// TIA Portal V19 export
FUNCTION_BLOCK "FlyingCarriage_FB"   // FB112, LAD
TITLE = FLYING SHEAR CARRIAGE
// stored: MemoryReserve 100, SetENOAutomatically false
   VAR_INPUT
      AreaInterface : "AreaInterface";
      ZSI : "udt_ZoneSafetyInterface";
      DSI : "udt_DeviceSafetyInterface";
      Drive { ExternalAccessible := 'False'; ExternalVisible := 'False'; ExternalWritable := 'False'} : "TAx_DriveInterface";
      CIn : "udt_FlyingCarriage_CIn";
      DataIn { ExternalAccessible := 'False'; ExternalVisible := 'False'; ExternalWritable := 'False'} : Struct
         Pb_Bkw : Bool;
         Pb_Fwd : Bool;
         Pb_Pos : Bool;
         Pb_Zero : Bool;
         Pb_PresetPos : Bool;
         Fbk_Fan : Bool;
      END_STRUCT;
      Config { ExternalAccessible := 'False'; ExternalVisible := 'False'; ExternalWritable := 'False'} : "udt_FlyingCarriage_Config";
   END_VAR
   VAR_OUTPUT
      MachineInterface : "MachineInterface";
      DataOut : Struct
         Fan : Bool;
         LP_ZeroOK : Bool;
      END_STRUCT;
   END_VAR
   VAR_IN_OUT
      TO_Carriage : TO_SynchronousAxis;
      TO_Master : TO_PositioningAxis;
      TO_ZeroChk : TO_MeasuringInput;
      Parameter : "udt_FlyingCarriage_Parameter";
      FsParameter : "udt_FsParameter";
   END_VAR
   VAR
      Warning : Struct
         NotAutReady : Bool := FALSE;
         ZeroChkRequest : Bool := FALSE;
         Axis : "TAx_Warnings";
      END_STRUCT;
      Alarm : Struct
         NotHomed : Bool := FALSE;
         ZeroChkFailed : Bool := FALSE;
         ZeroChk_NotCatched : Bool := FALSE;
         ZeroChk_NotReleased : Bool := FALSE;
         TargetPosition_OutOfRange : Bool := FALSE;
         Axis : "TAx_Alarms";
         ZeroChk : "TMeasuring_Alarms";
         Fan : "MotorAlr";
      END_STRUCT;
      Diag : Struct
         Ax : "TO_Diagnostic";
         ZeroChk : "TO_Diagnostic";   // 0 = No Msg; 1=Warning; 2= Fault
      END_STRUCT;
      COut : Struct
         Infeed_ReqON : Bool := FALSE;
         CtrlSafe : Bool := FALSE;
         Ax_InOperation : Bool := FALSE;
         Standstill : Bool := FALSE;
         CheckNext_Minus : Bool := FALSE;
         CheckNext_Plus : Bool := FALSE;
         PositioningDone : Bool := FALSE;
         InSynch : Bool := FALSE;
         ActualTargetPosAx : LReal := 0.0;
      END_STRUCT;
      HMI : Struct
         Pb_PresetPos : Bool := FALSE;
         PresetPosValue : LReal := 0.0;
         LastPositionDetect : LReal := 0.0;
         ManPosTarget : LReal;
         PositionNorm : Real;   // Normalized between 0.0 - 1.0
      END_STRUCT;
      Ax { S7_SetPoint := 'True'} : "FlyingShearAxis";
      MeasInp_ZeroChk { S7_SetPoint := 'True'} : "MeasuringInput";
      M_MotorFan : "Motor";
      tonDelayFanOff { S7_SetPoint := 'True'} : IEC_TIMER;
      tonDelayNoPendingCommands : IEC_TIMER;
      Sts : Struct
         IsStandstill : Bool;
         AlarmsPresence : Bool;
         WarningsPresence : Bool;
         DriveMessagesPresence : Bool;
         AxisMessagePresence : Bool;
         InOperatin : Bool;
         DriveParReadWriteDone : Bool;
         DriveMessagesReadDone : Bool;
         Gen_Condition : Bool;
         Bkw_Condition : Bool;
         Fwd_Condition : Bool;
         NoManCmd : Bool;
         Positioning_Condition : Bool;
         MotionRequestInNegativeDirection : Bool;
         MotionRequestInPositiveDirection : Bool;
         InPosition : Bool;
         AtHomePosition : Bool;
         Target_PosAx : LReal;
         MissingToTarget : LReal;
         ActualLimitMinus : LReal;
         ActualLimitPlus : LReal;
         ZeroChk_LastPositionDetect : LReal;
         ZeroChk_MeasInLastID : UInt;
      END_STRUCT;
      Ctrl : Struct
         RstAlarms : Bool;
         SafeMotion : Bool;
         StopDueDoorOpeningRequest : Bool;
         StopSafe : Bool;
         StopInPhase : Bool;
         StopProgrammed : Bool;
         StopAborting : Bool;
         ReadSLSParam : Bool;
         DriveParReadWrite_Exe : Bool;
         DriveMessageRead_Exe : Bool;
         Fan : Bool;
         Man_JogPosBkw : Bool;
         Man_JogPosFwd : Bool;
         Man_Pos : Bool;
         Man_Zero : Bool;
         Zero_Bkw : Bool;
         Zero_Fwd : Bool;
         Zero_Home : Bool;
         Man_Zero_Bkw : Bool;
         Man_Zero_Fwd : Bool;
         Man_Zero_Home : Bool;
         Man_PresetPosition : Bool;
         Aut_Zero : Bool;
         Aut_PosAbs : Bool;
         Aut_GearPos : Bool;
      END_STRUCT;
      AckRstAlarms : Bool := FALSE;
      Pb_Bkw_PEAux : Bool := FALSE;
      Pb_Fwd_PEAux : Bool := FALSE;
      Pb_Pos_PEAux : Bool := FALSE;
      Pb_Zero_PEAux : Bool := FALSE;
      Pb_PresetPos_PEAux : Bool := FALSE;
      ZeroChk_LastID : UInt := 0;
   END_VAR
   VAR_TEMP
      "NOP" : Bool;
      Pb_Bkw_PositiveEdge : Bool;
      Pb_Fwd_PositiveEdge : Bool;
      Pb_Pos_PositiveEdge : Bool;
      Pb_Zero_PositiveEdge : Bool;
      Pb_PresetPos_PositiveEdge : Bool;
      KP_FromProfilePrg : Real;
      KI_FromProfilePrg : Real;
      Delta_KP : Real;
      Delta_KI : Real;
      Delta_ChkZero : LReal;
      Jerk_Multi : LReal;
      Req : Bool;
   END_VAR
   VAR CONSTANT
      EXTENDED_SAFETY : Bool := FALSE;
      SLS_VEL : LReal := 3.0;
      DEFAULT_KV : LReal := 10.0;
      DEFAULT_KP : Real := 5.0;
      DEFAULT_KI : Real := 10.0;
      PAR_FLT : UInt := 0;
      PAR_ALM : UInt := 1;
      PAR_SLS : UInt := 2;
      PAR_KP : UInt := 3;
      PAR_KI : UInt := 4;
      DPS_IDLE : USInt := 0;
      DPS_REQUEST : USInt := 1;
      DPS_ACTIVE : USInt := 2;
      DPS_DONE : USInt := 10;
      DPS_ERROR : USInt := 11;
   END_VAR
   // MachineInterface.AutReady := FALSE;
   // MachineInterface.Aborting := FALSE;
   // MachineInterface.AckStopInPhase := FALSE;
   // MachineInterface.AckStopProgrammed := FALSE;
   // MachineInterface.MotionsStandStill := TRUE;
   // MachineInterface.AlarmsPresence := FALSE;
   // MachineInterface.WarningPresence := FALSE;
   VAR_TEMP   // added for the SCL form of the ladder/FBD networks
      _w1 : Bool;
      _w2 : Bool;
      _w3 : Bool;
      _w4 : Bool;
      _w5 : Bool;
   END_VAR
BEGIN

REGION Network 1: Push buttons positive edges
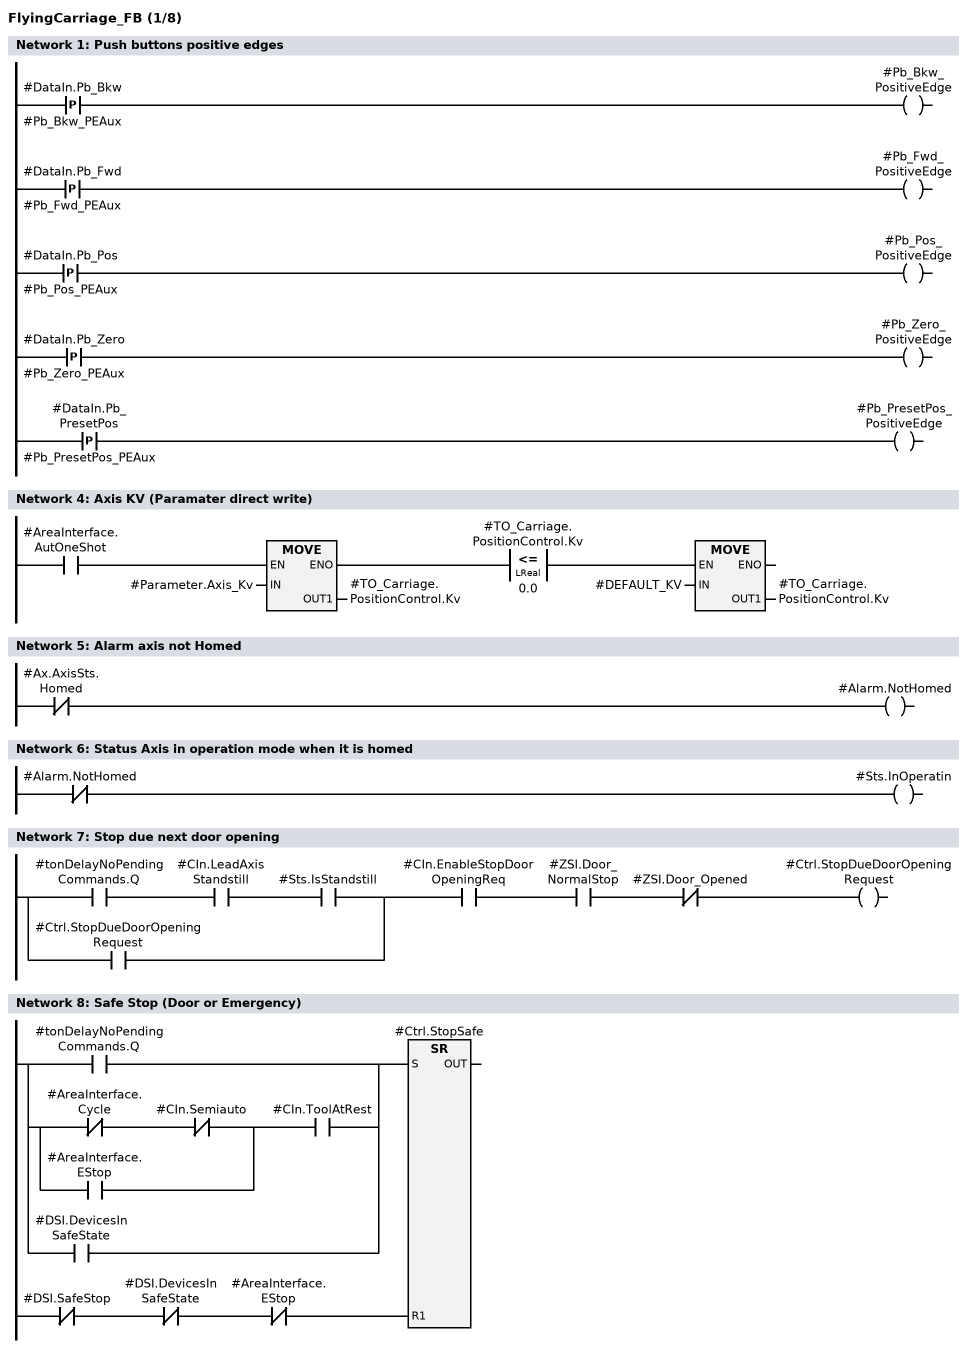
   RUNG wire#powerrail
      P_Contact(operand := #DataIn.Pb_Bkw, bit := #Pb_Bkw_PEAux)
      Coil( #Pb_Bkw_PositiveEdge )
   END_RUNG
   RUNG wire#powerrail
      P_Contact(operand := #DataIn.Pb_Fwd, bit := #Pb_Fwd_PEAux)
      Coil( #Pb_Fwd_PositiveEdge )
   END_RUNG
   RUNG wire#powerrail
      P_Contact(operand := #DataIn.Pb_Pos, bit := #Pb_Pos_PEAux)
      Coil( #Pb_Pos_PositiveEdge )
   END_RUNG
   RUNG wire#powerrail
      P_Contact(operand := #DataIn.Pb_Zero, bit := #Pb_Zero_PEAux)
      Coil( #Pb_Zero_PositiveEdge )
   END_RUNG
   RUNG wire#powerrail
      P_Contact(operand := #DataIn.Pb_PresetPos, bit := #Pb_PresetPos_PEAux)
      Coil( #Pb_PresetPos_PositiveEdge )
   END_RUNG
   // the same network as SCL:
   #_w1 := #DataIn.Pb_Bkw AND NOT #Pb_Bkw_PEAux;   // rising edge of #DataIn.Pb_Bkw
   #Pb_Bkw_PEAux := #DataIn.Pb_Bkw;
   #Pb_Bkw_PositiveEdge := #_w1;
   #_w2 := #DataIn.Pb_Fwd AND NOT #Pb_Fwd_PEAux;   // rising edge of #DataIn.Pb_Fwd
   #Pb_Fwd_PEAux := #DataIn.Pb_Fwd;
   #Pb_Fwd_PositiveEdge := #_w2;
   #_w3 := #DataIn.Pb_Pos AND NOT #Pb_Pos_PEAux;   // rising edge of #DataIn.Pb_Pos
   #Pb_Pos_PEAux := #DataIn.Pb_Pos;
   #Pb_Pos_PositiveEdge := #_w3;
   #_w4 := #DataIn.Pb_Zero AND NOT #Pb_Zero_PEAux;   // rising edge of #DataIn.Pb_Zero
   #Pb_Zero_PEAux := #DataIn.Pb_Zero;
   #Pb_Zero_PositiveEdge := #_w4;
   #_w5 := #DataIn.Pb_PresetPos AND NOT #Pb_PresetPos_PEAux;   // rising edge of #DataIn.Pb_PresetPos
   #Pb_PresetPos_PEAux := #DataIn.Pb_PresetPos;
   #Pb_PresetPos_PositiveEdge := #_w5;
END_REGION

REGION Network 2 (SCL): Reset alarms command
   #Ctrl.RstAlarms := #AreaInterface.RstAlarms AND NOT #AckRstAlarms; 
   #AckRstAlarms := #AreaInterface.RstAlarms;

   IF    #Ctrl.RstAlarms THEN

       #Warning.NotAutReady := FALSE;
       #Alarm.TargetPosition_OutOfRange := 
       #Alarm.ZeroChk_NotCatched :=
       #Alarm.ZeroChk_NotReleased :=
       #Alarm.ZeroChkFailed :=
       FALSE;

   END_IF;
END_REGION

REGION Network 3 (SCL): Controllo Zero
   // Zero Check Control
   #MeasInp_ZeroChk.MeasuringCtrl.MeasureEnable := 
           NOT #Alarm.NotHomed
           AND (NOT #Sts.IsStandstill OR #MeasInp_ZeroChk.MeasuringCtrl.MeasureEnable)
           AND NOT #AreaInterface.EStop
           AND NOT "Sys".SimulationDevice;        

   #MeasInp_ZeroChk.MeasuringCtrl.Mode := 0;
   #MeasInp_ZeroChk.MeasuringCtrl.Rst := #Ctrl.RstAlarms;

   // Main
   #MeasInp_ZeroChk(TO_Measuring:=#TO_ZeroChk,
                    Alarm := #Alarm.ZeroChk,
                    Diag := #Diag.ZeroChk);

   // Zero Check - Warning checking is request (each time EStop is rise up)
   IF #AreaInterface.EStop THEN 
       #ZeroChk_LastID :=
       #MeasInp_ZeroChk.Trigger_ID := 0;
       #Warning.ZeroChkRequest := TRUE;
   END_IF;

   IF (#AreaInterface.EStop OR  #ZeroChk_LastID = 0) AND NOT "Sys".SimulationDevice THEN
       #Warning.ZeroChkRequest  := TRUE;
   END_IF;



   // Zero Check - New position value detect
   IF  #MeasInp_ZeroChk.Trigger_ID <> #ZeroChk_LastID THEN
       #ZeroChk_LastID := #MeasInp_ZeroChk.Trigger_ID;
       #HMI.LastPositionDetect := #MeasInp_ZeroChk.MeasuringSts.MeasuringValue1;
       // Zero Check - Alarm Sensor position detect NOT match with deisred position
       IF ABS(#HMI.LastPositionDetect - #Parameter.ZeroChk_SensorPosition) > #Parameter.ZeroChk_PosTolerance THEN
           #Alarm.ZeroChkFailed := TRUE;
       ELSE
           #Warning.ZeroChkRequest := FALSE;
       END_IF;
   END_IF;
END_REGION

REGION Network 4: Axis KV (Paramater direct write)
   RUNG wire#powerrail
      Contact( #AreaInterface.AutOneShot )
      Move(in := #Parameter.Axis_Kv, out1 => #TO_Carriage.PositionControl.Kv)
      { S7_Templates := "SrcType := LReal" } LE_Contact(in1 := #TO_Carriage.PositionControl.Kv, in2 := 0.0)
      Move(in := #DEFAULT_KV, out1 => #TO_Carriage.PositionControl.Kv)
   END_RUNG
   // the same network as SCL:
   IF #AreaInterface.AutOneShot THEN #TO_Carriage.PositionControl.Kv := #Parameter.Axis_Kv; END_IF;
   IF #AreaInterface.AutOneShot AND (#TO_Carriage.PositionControl.Kv <= 0.0) THEN
       #TO_Carriage.PositionControl.Kv := #DEFAULT_KV;
   END_IF;
END_REGION

REGION Network 5: Alarm axis not Homed
   RUNG wire#powerrail
      I_Contact( #Ax.AxisSts.Homed )
      Coil( #Alarm.NotHomed )
   END_RUNG
   // the same network as SCL:
   #Alarm.NotHomed := NOT #Ax.AxisSts.Homed;
END_REGION

REGION Network 6: Status Axis in operation mode when it is homed
   RUNG wire#powerrail
      I_Contact( #Alarm.NotHomed )
      Coil( #Sts.InOperatin )
   END_RUNG
   // the same network as SCL:
   #Sts.InOperatin := NOT #Alarm.NotHomed;
END_REGION

REGION Network 7: Stop due next door opening
   RUNG wire#powerrail
      Contact( #tonDelayNoPendingCommands.Q )
      Contact( #CIn.LeadAxisStandstill )
      Contact( #Sts.IsStandstill )
      wire#w1
      Contact( #CIn.EnableStopDoorOpeningReq )
      Contact( #ZSI.Door_NormalStop )
      I_Contact( #ZSI.Door_Opened )
      Coil( #Ctrl.StopDueDoorOpeningRequest )
   END_RUNG
   RUNG wire#powerrail
      Contact( #Ctrl.StopDueDoorOpeningRequest )
   END_RUNG wire#w1
   // the same network as SCL:
   #Ctrl.StopDueDoorOpeningRequest := ((#tonDelayNoPendingCommands.Q AND #CIn.LeadAxisStandstill AND #Sts.IsStandstill) OR #Ctrl.StopDueDoorOpeningRequest) AND #CIn.EnableStopDoorOpeningReq AND #ZSI.Door_NormalStop AND NOT #ZSI.Door_Opened;
END_REGION

REGION Network 8: Safe Stop (Door or Emergency)
   RUNG wire#powerrail
      Contact( #tonDelayNoPendingCommands.Q )
      wire#w1
      S_SR(operand := #Ctrl.StopSafe, r1 := wire#w3)
   END_RUNG
   RUNG wire#powerrail
      I_Contact( #AreaInterface.Cycle )
      I_Contact( #CIn.Semiauto )
      wire#w2
      Contact( #CIn.ToolAtRest )
   END_RUNG wire#w1
   RUNG wire#powerrail
      Contact( #AreaInterface.EStop )
   END_RUNG wire#w2
   RUNG wire#powerrail
      Contact( #DSI.DevicesInSafeState )
   END_RUNG wire#w1
   RUNG wire#powerrail
      I_Contact( #DSI.SafeStop )
      I_Contact( #DSI.DevicesInSafeState )
      I_Contact( #AreaInterface.EStop )
   END_RUNG wire#w3
   // the same network as SCL:
   IF #tonDelayNoPendingCommands.Q OR (((NOT #AreaInterface.Cycle AND NOT #CIn.Semiauto) OR #AreaInterface.EStop) AND #CIn.ToolAtRest) OR #DSI.DevicesInSafeState THEN
       #Ctrl.StopSafe := TRUE;   // SR flip-flop
   END_IF;
   IF NOT #DSI.SafeStop AND NOT #DSI.DevicesInSafeState AND NOT #AreaInterface.EStop THEN
       #Ctrl.StopSafe := FALSE;
   END_IF;
END_REGION

REGION Network 9: Safe Motion
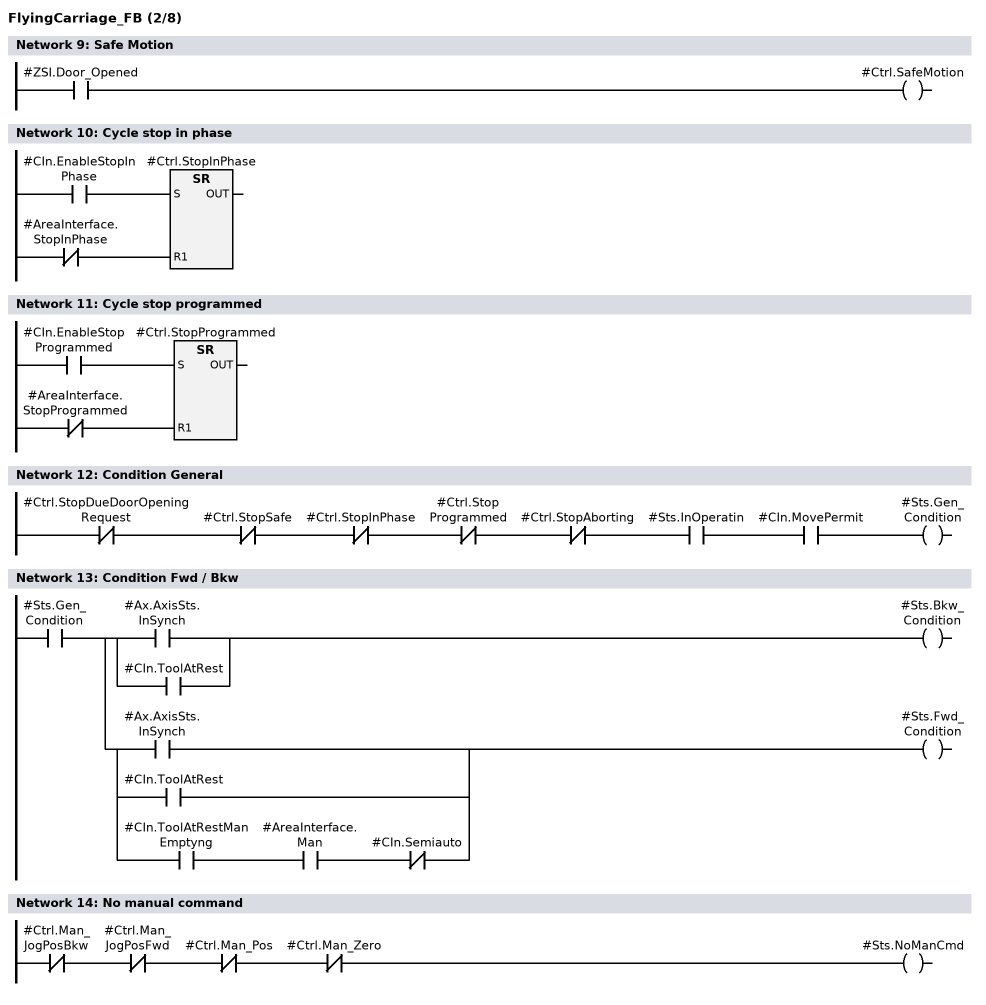
   RUNG wire#powerrail
      Contact( #ZSI.Door_Opened )
      Coil( #Ctrl.SafeMotion )
   END_RUNG
   // the same network as SCL:
   #Ctrl.SafeMotion := #ZSI.Door_Opened;
END_REGION

REGION Network 10: Cycle stop in phase
   RUNG wire#powerrail
      Contact( #CIn.EnableStopInPhase )
      S_SR(operand := #Ctrl.StopInPhase, r1 := wire#w1)
   END_RUNG
   RUNG wire#powerrail
      I_Contact( #AreaInterface.StopInPhase )
   END_RUNG wire#w1
   // the same network as SCL:
   IF #CIn.EnableStopInPhase THEN
       #Ctrl.StopInPhase := TRUE;   // SR flip-flop
   END_IF;
   IF NOT #AreaInterface.StopInPhase THEN #Ctrl.StopInPhase := FALSE; END_IF;
END_REGION

REGION Network 11: Cycle stop programmed
   RUNG wire#powerrail
      Contact( #CIn.EnableStopProgrammed )
      S_SR(operand := #Ctrl.StopProgrammed, r1 := wire#w1)
   END_RUNG
   RUNG wire#powerrail
      I_Contact( #AreaInterface.StopProgrammed )
   END_RUNG wire#w1
   // the same network as SCL:
   IF #CIn.EnableStopProgrammed THEN
       #Ctrl.StopProgrammed := TRUE;   // SR flip-flop
   END_IF;
   IF NOT #AreaInterface.StopProgrammed THEN #Ctrl.StopProgrammed := FALSE; END_IF;
END_REGION

REGION Network 12: Condition General
   RUNG wire#powerrail
      I_Contact( #Ctrl.StopDueDoorOpeningRequest )
      I_Contact( #Ctrl.StopSafe )
      I_Contact( #Ctrl.StopInPhase )
      I_Contact( #Ctrl.StopProgrammed )
      I_Contact( #Ctrl.StopAborting )
      Contact( #Sts.InOperatin )
      Contact( #CIn.MovePermit )
      Coil( #Sts.Gen_Condition )
   END_RUNG
   // the same network as SCL:
   #Sts.Gen_Condition := NOT #Ctrl.StopDueDoorOpeningRequest AND NOT #Ctrl.StopSafe AND NOT #Ctrl.StopInPhase AND NOT #Ctrl.StopProgrammed AND NOT #Ctrl.StopAborting AND #Sts.InOperatin AND #CIn.MovePermit;
END_REGION

REGION Network 13: Condition Fwd / Bkw
   RUNG wire#powerrail
      Contact( #Sts.Gen_Condition )
      wire#w1
      Contact( #Ax.AxisSts.InSynch )
      wire#w2
      Coil( #Sts.Bkw_Condition )
   END_RUNG
   RUNG wire#w1
      Contact( #CIn.ToolAtRest )
   END_RUNG wire#w2
   RUNG wire#w1
      Contact( #Ax.AxisSts.InSynch )
      wire#w3
      Coil( #Sts.Fwd_Condition )
   END_RUNG
   RUNG wire#w1
      Contact( #CIn.ToolAtRest )
   END_RUNG wire#w3
   RUNG wire#w1
      Contact( #CIn.ToolAtRestManEmptyng )
      Contact( #AreaInterface.Man )
      I_Contact( #CIn.Semiauto )
   END_RUNG wire#w3
   // the same network as SCL:
   #Sts.Bkw_Condition := #Sts.Gen_Condition AND (#Ax.AxisSts.InSynch OR #CIn.ToolAtRest);
   #Sts.Fwd_Condition := #Sts.Gen_Condition AND (#Ax.AxisSts.InSynch OR #CIn.ToolAtRest OR (#CIn.ToolAtRestManEmptyng AND #AreaInterface.Man AND NOT #CIn.Semiauto));
END_REGION

REGION Network 14: No manual command
   RUNG wire#powerrail
      I_Contact( #Ctrl.Man_JogPosBkw )
      I_Contact( #Ctrl.Man_JogPosFwd )
      I_Contact( #Ctrl.Man_Pos )
      I_Contact( #Ctrl.Man_Zero )
      Coil( #Sts.NoManCmd )
   END_RUNG
   // the same network as SCL:
   #Sts.NoManCmd := NOT #Ctrl.Man_JogPosBkw AND NOT #Ctrl.Man_JogPosFwd AND NOT #Ctrl.Man_Pos AND NOT #Ctrl.Man_Zero;
END_REGION

REGION Network 15: Man Jog Bkw / Fwd using positioning / Preset position
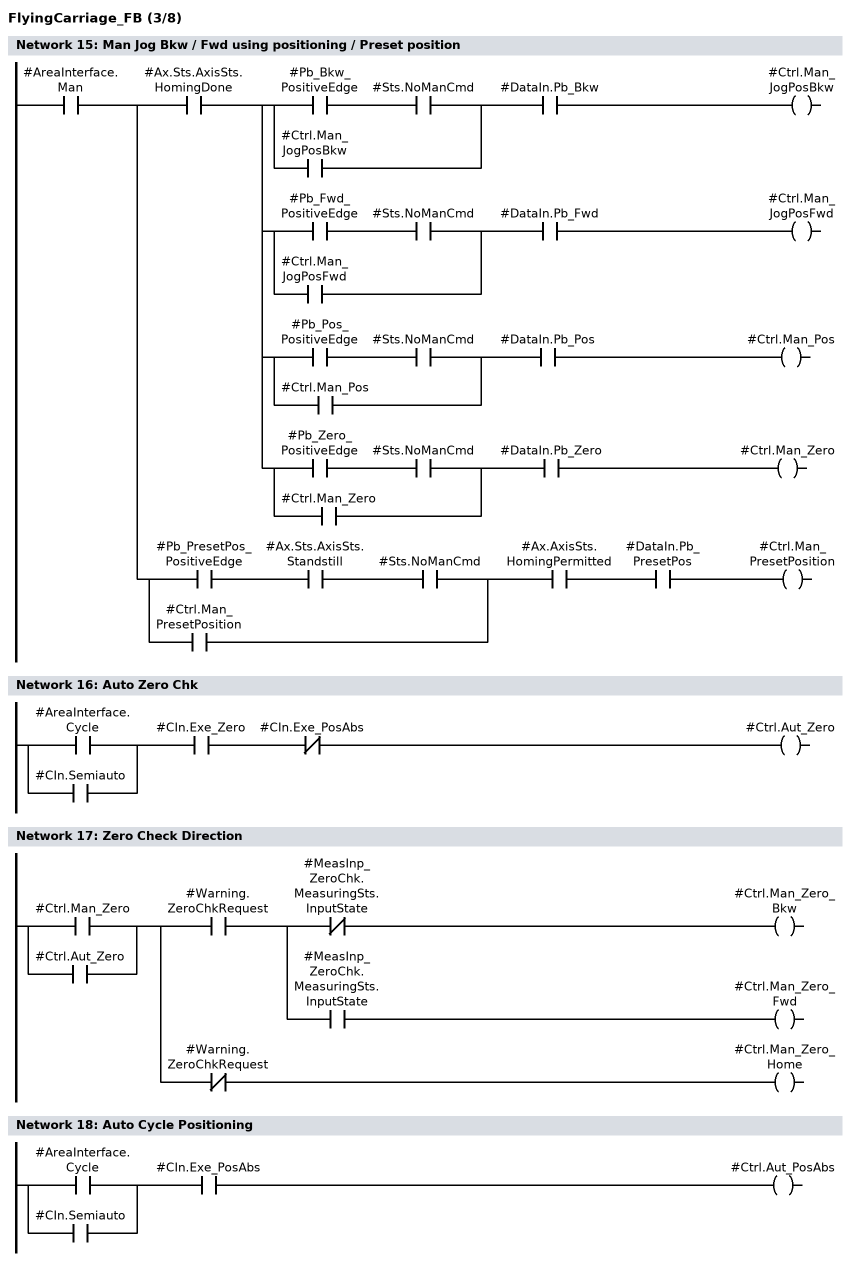
   RUNG wire#powerrail
      Contact( #AreaInterface.Man )
      wire#w1
      Contact( #Ax.Sts.AxisSts.HomingDone )
      wire#w2
      Contact( #Pb_Bkw_PositiveEdge )
      Contact( #Sts.NoManCmd )
      wire#w3
      Contact( #DataIn.Pb_Bkw )
      Coil( #Ctrl.Man_JogPosBkw )
   END_RUNG
   RUNG wire#w2
      Contact( #Ctrl.Man_JogPosBkw )
   END_RUNG wire#w3
   RUNG wire#w2
      Contact( #Pb_Fwd_PositiveEdge )
      Contact( #Sts.NoManCmd )
      wire#w4
      Contact( #DataIn.Pb_Fwd )
      Coil( #Ctrl.Man_JogPosFwd )
   END_RUNG
   RUNG wire#w2
      Contact( #Ctrl.Man_JogPosFwd )
   END_RUNG wire#w4
   RUNG wire#w2
      Contact( #Pb_Pos_PositiveEdge )
      Contact( #Sts.NoManCmd )
      wire#w5
      Contact( #DataIn.Pb_Pos )
      Coil( #Ctrl.Man_Pos )
   END_RUNG
   RUNG wire#w2
      Contact( #Ctrl.Man_Pos )
   END_RUNG wire#w5
   RUNG wire#w2
      Contact( #Pb_Zero_PositiveEdge )
      Contact( #Sts.NoManCmd )
      wire#w6
      Contact( #DataIn.Pb_Zero )
      Coil( #Ctrl.Man_Zero )
   END_RUNG
   RUNG wire#w2
      Contact( #Ctrl.Man_Zero )
   END_RUNG wire#w6
   RUNG wire#w1
      Contact( #Pb_PresetPos_PositiveEdge )
      Contact( #Ax.Sts.AxisSts.Standstill )
      Contact( #Sts.NoManCmd )
      wire#w7
      Contact( #Ax.AxisSts.HomingPermitted )
      Contact( #DataIn.Pb_PresetPos )
      Coil( #Ctrl.Man_PresetPosition )
   END_RUNG
   RUNG wire#w1
      Contact( #Ctrl.Man_PresetPosition )
   END_RUNG wire#w7
   // the same network as SCL:
   #_w1 := #AreaInterface.Man AND #Ax.Sts.AxisSts.HomingDone;
   #Ctrl.Man_JogPosBkw := #_w1 AND ((#Pb_Bkw_PositiveEdge AND #Sts.NoManCmd) OR #Ctrl.Man_JogPosBkw) AND #DataIn.Pb_Bkw;
   #Ctrl.Man_JogPosFwd := #_w1 AND ((#Pb_Fwd_PositiveEdge AND #Sts.NoManCmd) OR #Ctrl.Man_JogPosFwd) AND #DataIn.Pb_Fwd;
   #Ctrl.Man_Pos := #_w1 AND ((#Pb_Pos_PositiveEdge AND #Sts.NoManCmd) OR #Ctrl.Man_Pos) AND #DataIn.Pb_Pos;
   #Ctrl.Man_Zero := #_w1 AND ((#Pb_Zero_PositiveEdge AND #Sts.NoManCmd) OR #Ctrl.Man_Zero) AND #DataIn.Pb_Zero;
   #Ctrl.Man_PresetPosition := #AreaInterface.Man AND ((#Pb_PresetPos_PositiveEdge AND #Ax.Sts.AxisSts.Standstill AND #Sts.NoManCmd) OR #Ctrl.Man_PresetPosition) AND #Ax.AxisSts.HomingPermitted AND #DataIn.Pb_PresetPos;
END_REGION

REGION Network 16: Auto Zero Chk
   RUNG wire#powerrail
      Contact( #AreaInterface.Cycle )
      wire#w1
      Contact( #CIn.Exe_Zero )
      I_Contact( #CIn.Exe_PosAbs )
      Coil( #Ctrl.Aut_Zero )
   END_RUNG
   RUNG wire#powerrail
      Contact( #CIn.Semiauto )
   END_RUNG wire#w1
   // the same network as SCL:
   #Ctrl.Aut_Zero := (#AreaInterface.Cycle OR #CIn.Semiauto) AND #CIn.Exe_Zero AND NOT #CIn.Exe_PosAbs;
END_REGION

REGION Network 17: Zero Check Direction
   RUNG wire#powerrail
      Contact( #Ctrl.Man_Zero )
      wire#w1
      Contact( #Warning.ZeroChkRequest )
      wire#w2
      I_Contact( #MeasInp_ZeroChk.MeasuringSts.InputState )
      Coil( #Ctrl.Man_Zero_Bkw )
   END_RUNG
   RUNG wire#powerrail
      Contact( #Ctrl.Aut_Zero )
   END_RUNG wire#w1
   RUNG wire#w2
      Contact( #MeasInp_ZeroChk.MeasuringSts.InputState )
      Coil( #Ctrl.Man_Zero_Fwd )
   END_RUNG
   RUNG wire#w1
      I_Contact( #Warning.ZeroChkRequest )
      Coil( #Ctrl.Man_Zero_Home )
   END_RUNG
   // the same network as SCL:
   #_w1 := #Ctrl.Man_Zero OR #Ctrl.Aut_Zero;
   #_w2 := #_w1 AND #Warning.ZeroChkRequest;
   #Ctrl.Man_Zero_Bkw := #_w2 AND NOT #MeasInp_ZeroChk.MeasuringSts.InputState;
   #Ctrl.Man_Zero_Fwd := #_w2 AND #MeasInp_ZeroChk.MeasuringSts.InputState;
   #Ctrl.Man_Zero_Home := #_w1 AND NOT #Warning.ZeroChkRequest;
END_REGION

REGION Network 18: Auto Cycle Positioning
   RUNG wire#powerrail
      Contact( #AreaInterface.Cycle )
      wire#w1
      Contact( #CIn.Exe_PosAbs )
      Coil( #Ctrl.Aut_PosAbs )
   END_RUNG
   RUNG wire#powerrail
      Contact( #CIn.Semiauto )
   END_RUNG wire#w1
   // the same network as SCL:
   #Ctrl.Aut_PosAbs := (#AreaInterface.Cycle OR #CIn.Semiauto) AND #CIn.Exe_PosAbs;
END_REGION

REGION Network 19: Axis Sowftware Limits
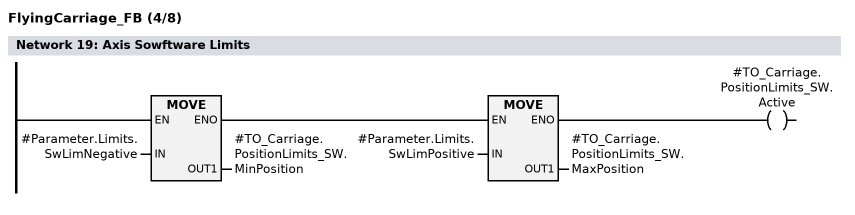
   RUNG wire#powerrail
      Move(in := #Parameter.Limits.SwLimNegative, out1 => #TO_Carriage.PositionLimits_SW.MinPosition)
      Move(in := #Parameter.Limits.SwLimPositive, out1 => #TO_Carriage.PositionLimits_SW.MaxPosition)
      Coil( #TO_Carriage.PositionLimits_SW.Active )
   END_RUNG
   // the same network as SCL:
   #TO_Carriage.PositionLimits_SW.MinPosition := #Parameter.Limits.SwLimNegative;
   #TO_Carriage.PositionLimits_SW.MaxPosition := #Parameter.Limits.SwLimPositive;
   #TO_Carriage.PositionLimits_SW.Active := TRUE;
END_REGION

REGION Network 20 (SCL): Actual position Limits
   #Sts.ActualLimitMinus := #TO_Carriage.PositionLimits_SW.MinPosition + #Parameter.PosTolerance;
   #Sts.ActualLimitPlus := #TO_Carriage.PositionLimits_SW.MaxPosition - #Parameter.PosTolerance;
END_REGION

REGION Network 21 (SCL): Target Position & Positioning condition
   // Target Position

   IF #AreaInterface.Cycle OR (#CIn.Semiauto AND NOT #CIn.Exe_Zero) THEN
       #Sts.Target_PosAx := #CIn.PosAbs_TargetPosAx;
       #HMI.ManPosTarget := #CIn.PosAbs_TargetPosAx;
   ELSIF #Ctrl.Man_Pos THEN
       #Sts.Target_PosAx := #HMI.ManPosTarget;
   ELSIF #Ctrl.Man_JogPosBkw OR #Ctrl.Man_Zero_Bkw THEN
       #Sts.Target_PosAx := #Sts.ActualLimitMinus;
   ELSIF #Ctrl.Man_Zero_Home THEN
       #Sts.Target_PosAx := #FsParameter.Positions.HomePosition;
   ELSIF #Ctrl.Man_JogPosFwd OR #Ctrl.Man_Zero_Fwd THEN
       #Sts.Target_PosAx := #Sts.ActualLimitPlus;
   END_IF;

   #Ax.AxisCtrl.MoveAbsTarget := #Sts.Target_PosAx;

   // At Home Position
   #Sts.AtHomePosition := ABS(#FsParameter.Positions.HomePosition - #TO_Carriage.ActualPosition) < #Parameter.PosTolerance
   AND NOT #Warning.ZeroChkRequest;

   // Positioning Condition

   #Sts.MissingToTarget := #Sts.Target_PosAx - #TO_Carriage.ActualPosition;

   #Sts.Positioning_Condition := FALSE;
   #Sts.InPosition := FALSE;


   IF ABS(#Sts.MissingToTarget) < #Parameter.PosTolerance THEN

       #Sts.Positioning_Condition := TRUE;
       #Sts.InPosition := TRUE;

       IF #Ctrl.Man_Zero_Bkw THEN
           #Alarm.ZeroChk_NotCatched := TRUE;
       END_IF;
       IF  #Ctrl.Man_Zero_Fwd THEN
           #Alarm.ZeroChk_NotReleased := TRUE;
       END_IF;

   ELSIF #Sts.MissingToTarget > 0.0 AND #Sts.Fwd_Condition AND #Ax.AxisSts.MoveAbsPermitted THEN

       #Sts.Positioning_Condition := TRUE;

   ELSIF #Sts.MissingToTarget < 0.0 AND #Sts.Bkw_Condition AND #Ax.AxisSts.MoveAbsPermitted THEN

       #Sts.Positioning_Condition := TRUE;
   END_IF;

   IF ((#Sts.Target_PosAx > #TO_Carriage.PositionLimits_SW.MaxPosition) OR
       (#Sts.Target_PosAx < #TO_Carriage.PositionLimits_SW.MinPosition))
       AND (#Ctrl.Aut_PosAbs OR #Ctrl.Man_Pos) THEN
       #Sts.Positioning_Condition := FALSE;
       #Alarm.TargetPosition_OutOfRange := TRUE;
   END_IF;
END_REGION

REGION Network 22 (SCL): Target Velocity / Acceleration / Deceleration / Jerk
   // Jerk Multiplier 
   #Jerk_Multi := SEL(G := #TO_Carriage.Units.VelocityUnit = 1524, IN0 := 1000.0, IN1 := 1.0);

   // Target Velocity
   IF #AreaInterface.Man OR #CIn.Semiauto THEN
       #Ax.AxisCtrl.Velocity := #Parameter.Man.Vel;


   ELSIF #Ctrl.Aut_PosAbs THEN

        #Ax.AxisCtrl.Velocity := #CIn.PosAbs_Vel;
   ELSE

     #Ax.AxisCtrl.Velocity := 0.0;


   END_IF;


   // Target Acc/Dec/Jerk
   // IF   #Ctrl.Man_JogPosBkw OR #Ctrl.Man_JogPosFwd OR #Ctrl.Man_Pos THEN
   IF #AreaInterface.Man THEN

       #Ax.AxisCtrl.Acceleration := #Parameter.Man.Acc;
       #Ax.AxisCtrl.Deceleration := #Parameter.Man.Dec;
       #Ax.AxisCtrl.Jerk := #Parameter.Man.Jerk * #Jerk_Multi;

   ELSIF   #AreaInterface.Cycle THEN

       #Ax.AxisCtrl.Acceleration := #CIn.PosAbs_Acc; 
       #Ax.AxisCtrl.Deceleration := #CIn.PosAbs_Dec;
       #Ax.AxisCtrl.Jerk := #CIn.PosAbs_Jerk * #Jerk_Multi;

   END_IF;

   // Default dynamics values
   IF      #Ax.AxisCtrl.Acceleration <= 0 OR #Ax.AxisCtrl.Deceleration <= 0 THEN

       #Ax.AxisCtrl.Acceleration := #Parameter.Aut.Acc;
       #Ax.AxisCtrl.Deceleration := #Parameter.Aut.Dec;
       #Ax.AxisCtrl.Jerk := #Parameter.Aut.Jerk * #Jerk_Multi;
   END_IF; 


   // Dynamics if Safe motion
   IF #Ctrl.SafeMotion OR #Ctrl.StopSafe OR #Warning.ZeroChkRequest THEN
       #Ax.AxisCtrl.Velocity := MIN(IN1 := #Ax.AxisCtrl.Velocity, IN2 := #Config.SLS_VEL);
       (*
       #Ax.AxisCtrl.Acceleration := #Config.SLS_ACC;
       #Ax.AxisCtrl.Deceleration := #Config.SLS_DEC;
       #Ax.AxisCtrl.Jerk := #Config.SLS_JERK * #Jerk_Multi; *)
   END_IF;
END_REGION

REGION Network 23: Axis controls
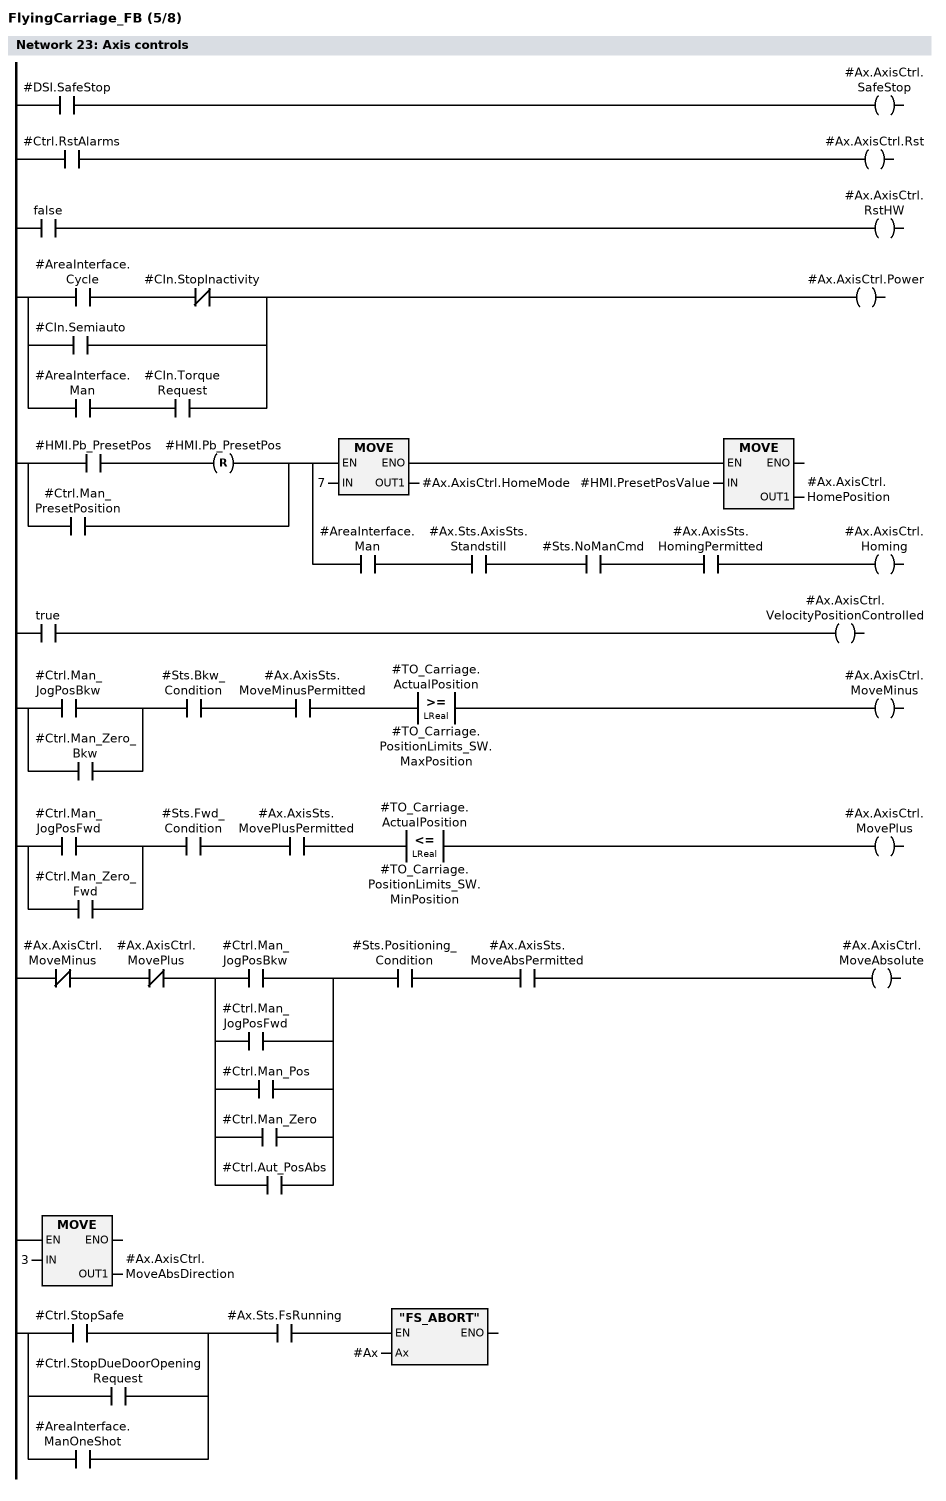
   RUNG wire#powerrail
      Contact( #DSI.SafeStop )
      Coil( #Ax.AxisCtrl.SafeStop )
   END_RUNG
   RUNG wire#powerrail
      Contact( #Ctrl.RstAlarms )
      Coil( #Ax.AxisCtrl.Rst )
   END_RUNG
   RUNG wire#powerrail
      Contact( false )
      Coil( #Ax.AxisCtrl.RstHW )
   END_RUNG
   RUNG wire#powerrail
      Contact( #AreaInterface.Cycle )
      I_Contact( #CIn.StopInactivity )
      wire#w1
      Coil( #Ax.AxisCtrl.Power )
   END_RUNG
   RUNG wire#powerrail
      Contact( #CIn.Semiauto )
   END_RUNG wire#w1
   RUNG wire#powerrail
      Contact( #AreaInterface.Man )
      Contact( #CIn.TorqueRequest )
   END_RUNG wire#w1
   RUNG wire#powerrail
      Contact( #HMI.Pb_PresetPos )
      R_Coil( #HMI.Pb_PresetPos )
      wire#w2
      Move(in := 7, out1 => #Ax.AxisCtrl.HomeMode)
      Move(in := #HMI.PresetPosValue, out1 => #Ax.AxisCtrl.HomePosition)
   END_RUNG
   RUNG wire#powerrail
      Contact( #Ctrl.Man_PresetPosition )
   END_RUNG wire#w2
   RUNG wire#w2
      Contact( #AreaInterface.Man )
      Contact( #Ax.Sts.AxisSts.Standstill )
      Contact( #Sts.NoManCmd )
      Contact( #Ax.AxisSts.HomingPermitted )
      Coil( #Ax.AxisCtrl.Homing )
   END_RUNG
   RUNG wire#powerrail
      Contact( true )
      Coil( #Ax.AxisCtrl.VelocityPositionControlled )
   END_RUNG
   RUNG wire#powerrail
      Contact( #Ctrl.Man_JogPosBkw )
      wire#w3
      Contact( #Sts.Bkw_Condition )
      Contact( #Ax.AxisSts.MoveMinusPermitted )
      { S7_Templates := "SrcType := LReal" } GE_Contact(in1 := #TO_Carriage.ActualPosition, in2 := #TO_Carriage.PositionLimits_SW.MaxPosition)
      Coil( #Ax.AxisCtrl.MoveMinus )
   END_RUNG
   RUNG wire#powerrail
      Contact( #Ctrl.Man_Zero_Bkw )
   END_RUNG wire#w3
   RUNG wire#powerrail
      Contact( #Ctrl.Man_JogPosFwd )
      wire#w4
      Contact( #Sts.Fwd_Condition )
      Contact( #Ax.AxisSts.MovePlusPermitted )
      { S7_Templates := "SrcType := LReal" } LE_Contact(in1 := #TO_Carriage.ActualPosition, in2 := #TO_Carriage.PositionLimits_SW.MinPosition)
      Coil( #Ax.AxisCtrl.MovePlus )
   END_RUNG
   RUNG wire#powerrail
      Contact( #Ctrl.Man_Zero_Fwd )
   END_RUNG wire#w4
   RUNG wire#powerrail
      I_Contact( #Ax.AxisCtrl.MoveMinus )
      I_Contact( #Ax.AxisCtrl.MovePlus )
      wire#w5
      Contact( #Ctrl.Man_JogPosBkw )
      wire#w6
      Contact( #Sts.Positioning_Condition )
      Contact( #Ax.AxisSts.MoveAbsPermitted )
      Coil( #Ax.AxisCtrl.MoveAbsolute )
   END_RUNG
   RUNG wire#w5
      Contact( #Ctrl.Man_JogPosFwd )
   END_RUNG wire#w6
   RUNG wire#w5
      Contact( #Ctrl.Man_Pos )
   END_RUNG wire#w6
   RUNG wire#w5
      Contact( #Ctrl.Man_Zero )
   END_RUNG wire#w6
   RUNG wire#w5
      Contact( #Ctrl.Aut_PosAbs )
   END_RUNG wire#w6
   RUNG wire#powerrail
      Move(in := 3, out1 => #Ax.AxisCtrl.MoveAbsDirection)
   END_RUNG
   RUNG wire#powerrail
      Contact( #Ctrl.StopSafe )
      wire#w7
      Contact( #Ax.Sts.FsRunning )
      "FS_ABORT"(Ax := #Ax)
   END_RUNG
   RUNG wire#powerrail
      Contact( #Ctrl.StopDueDoorOpeningRequest )
   END_RUNG wire#w7
   RUNG wire#powerrail
      Contact( #AreaInterface.ManOneShot )
   END_RUNG wire#w7
   // the same network as SCL:
   #Ax.AxisCtrl.SafeStop := #DSI.SafeStop;
   #Ax.AxisCtrl.Rst := #Ctrl.RstAlarms;
   #Ax.AxisCtrl.RstHW := false;
   #Ax.AxisCtrl.Power := (#AreaInterface.Cycle AND NOT #CIn.StopInactivity) OR #CIn.Semiauto OR (#AreaInterface.Man AND #CIn.TorqueRequest);
   #_w1 := #HMI.Pb_PresetPos;
   IF #_w1 THEN #HMI.Pb_PresetPos := FALSE; END_IF;
   #_w2 := #_w1 OR #Ctrl.Man_PresetPosition;
   IF #_w2 THEN
       #Ax.AxisCtrl.HomeMode := 7;
       #Ax.AxisCtrl.HomePosition := #HMI.PresetPosValue;
   END_IF;
   #Ax.AxisCtrl.Homing := #_w2 AND #AreaInterface.Man AND #Ax.Sts.AxisSts.Standstill AND #Sts.NoManCmd AND #Ax.AxisSts.HomingPermitted;
   #Ax.AxisCtrl.VelocityPositionControlled := true;
   #Ax.AxisCtrl.MoveMinus := (#Ctrl.Man_JogPosBkw OR #Ctrl.Man_Zero_Bkw) AND #Sts.Bkw_Condition AND #Ax.AxisSts.MoveMinusPermitted AND (#TO_Carriage.ActualPosition >= #TO_Carriage.PositionLimits_SW.MaxPosition);
   #Ax.AxisCtrl.MovePlus := (#Ctrl.Man_JogPosFwd OR #Ctrl.Man_Zero_Fwd) AND #Sts.Fwd_Condition AND #Ax.AxisSts.MovePlusPermitted AND (#TO_Carriage.ActualPosition <= #TO_Carriage.PositionLimits_SW.MinPosition);
   #Ax.AxisCtrl.MoveAbsolute := NOT #Ax.AxisCtrl.MoveMinus AND NOT #Ax.AxisCtrl.MovePlus AND (#Ctrl.Man_JogPosBkw OR #Ctrl.Man_JogPosFwd OR #Ctrl.Man_Pos OR #Ctrl.Man_Zero OR #Ctrl.Aut_PosAbs) AND #Sts.Positioning_Condition AND #Ax.AxisSts.MoveAbsPermitted;
   #Ax.AxisCtrl.MoveAbsDirection := 3;
   IF (#Ctrl.StopSafe OR #Ctrl.StopDueDoorOpeningRequest OR #AreaInterface.ManOneShot) AND #Ax.Sts.FsRunning THEN
       "FS_ABORT"(Ax := #Ax);
   END_IF;
END_REGION

REGION Network 24: Axis manager
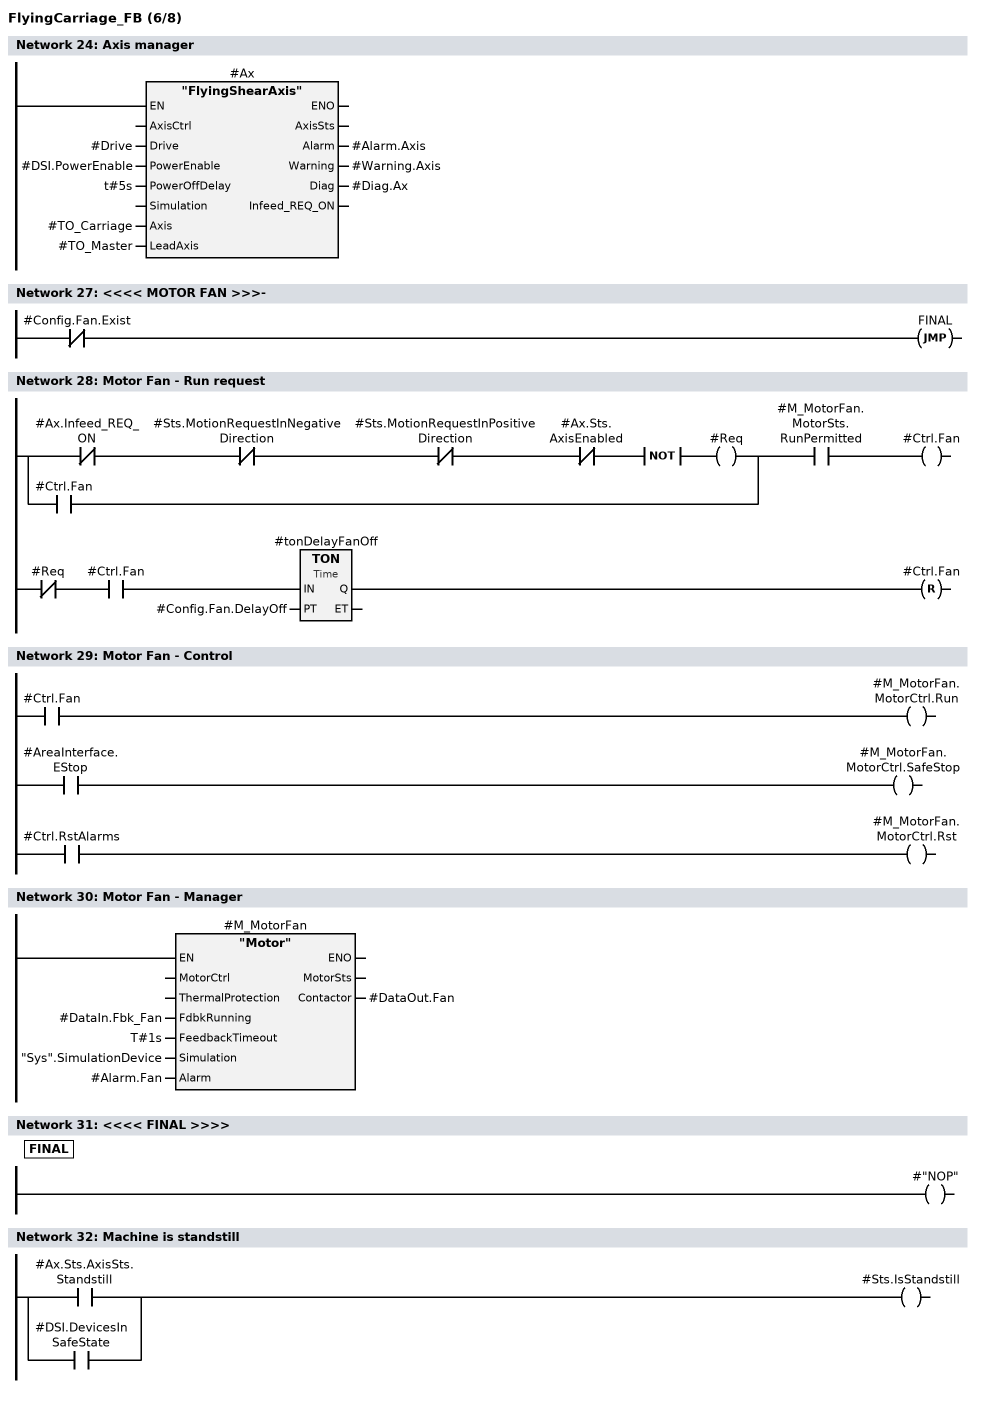
   RUNG wire#powerrail
      #Ax(AxisCtrl :=, Drive := #Drive, PowerEnable := #DSI.PowerEnable, PowerOffDelay := t#5s, Simulation :=, Axis := #TO_Carriage, LeadAxis := #TO_Master, AxisSts =>, Alarm => #Alarm.Axis, Warning => #Warning.Axis, Diag => #Diag.Ax, Infeed_REQ_ON =>)
   END_RUNG
   // the same network as SCL:
   #Ax(Drive := #Drive,   // "FlyingShearAxis"
       PowerEnable := #DSI.PowerEnable,
       PowerOffDelay := t#5s,
       Axis := #TO_Carriage,
       LeadAxis := #TO_Master,
       Alarm => #Alarm.Axis,
       Warning => #Warning.Axis,
       Diag => #Diag.Ax);
END_REGION

REGION Network 25 (SCL): Motion request in negative direction
   IF (#Ctrl.Aut_PosAbs OR #Ctrl.Man_Pos OR #Ctrl.Man_JogPosBkw OR #Ctrl.Man_Zero OR #Ctrl.Aut_Zero)
       AND
       #Sts.MissingToTarget < - #Parameter.PosTolerance THEN
       #Sts.MotionRequestInNegativeDirection := TRUE;
   ELSE
       #Sts.MotionRequestInNegativeDirection := FALSE;
   END_IF;
END_REGION

REGION Network 26 (SCL): Motion request in poisitive direction
   IF #Ctrl.Aut_GearPos THEN
       #Sts.MotionRequestInPositiveDirection := TRUE;

   ELSIF (#Ctrl.Man_JogPosFwd OR #Ctrl.Aut_PosAbs OR #Ctrl.Man_Pos OR #Ctrl.Zero_Fwd OR #Ctrl.Man_Zero OR #Ctrl.Aut_Zero)
       AND
       #Sts.MissingToTarget > #Parameter.PosTolerance  THEN
       #Sts.MotionRequestInPositiveDirection := TRUE;
   ELSE
       #Sts.MotionRequestInPositiveDirection := FALSE;
   END_IF;
END_REGION

REGION Network 27: <<<< MOTOR FAN >>>-
   RUNG wire#powerrail
      I_Contact( #Config.Fan.Exist )
      JumpCoil( FINAL )
   END_RUNG
   // the same network as SCL:
   IF NOT #Config.Fan.Exist THEN GOTO FINAL; END_IF;
END_REGION

REGION Network 28: Motor Fan - Run request
   RUNG wire#powerrail
      I_Contact( #Ax.Infeed_REQ_ON )
      I_Contact( #Sts.MotionRequestInNegativeDirection )
      I_Contact( #Sts.MotionRequestInPositiveDirection )
      I_Contact( #Ax.Sts.AxisEnabled )
      Not()
      Coil( #Req )
      wire#w1
      Contact( #M_MotorFan.MotorSts.RunPermitted )
      Coil( #Ctrl.Fan )
   END_RUNG
   RUNG wire#powerrail
      Contact( #Ctrl.Fan )
   END_RUNG wire#w1
   RUNG wire#powerrail
      I_Contact( #Req )
      Contact( #Ctrl.Fan )
      { S7_Templates := "time_type := Time" } #tonDelayFanOff.TON(pt := #Config.Fan.DelayOff, et =>)
      R_Coil( #Ctrl.Fan )
   END_RUNG
   // the same network as SCL:
   #Req := NOT (NOT #Ax.Infeed_REQ_ON AND NOT #Sts.MotionRequestInNegativeDirection AND NOT #Sts.MotionRequestInPositiveDirection AND NOT #Ax.Sts.AxisEnabled);
   #Ctrl.Fan := (#Req OR #Ctrl.Fan) AND #M_MotorFan.MotorSts.RunPermitted;
   #tonDelayFanOff.TON(IN := NOT #Req AND #Ctrl.Fan, PT := #Config.Fan.DelayOff);
   IF #tonDelayFanOff.Q THEN #Ctrl.Fan := FALSE; END_IF;
END_REGION

REGION Network 29: Motor Fan - Control
   RUNG wire#powerrail
      Contact( #Ctrl.Fan )
      Coil( #M_MotorFan.MotorCtrl.Run )
   END_RUNG
   RUNG wire#powerrail
      Contact( #AreaInterface.EStop )
      Coil( #M_MotorFan.MotorCtrl.SafeStop )
   END_RUNG
   RUNG wire#powerrail
      Contact( #Ctrl.RstAlarms )
      Coil( #M_MotorFan.MotorCtrl.Rst )
   END_RUNG
   // the same network as SCL:
   #M_MotorFan.MotorCtrl.Run := #Ctrl.Fan;
   #M_MotorFan.MotorCtrl.SafeStop := #AreaInterface.EStop;
   #M_MotorFan.MotorCtrl.Rst := #Ctrl.RstAlarms;
END_REGION

REGION Network 30: Motor Fan - Manager
   RUNG wire#powerrail
      #M_MotorFan(MotorCtrl :=, ThermalProtection :=, FdbkRunning := #DataIn.Fbk_Fan, FeedbackTimeout := T#1s, Simulation := "Sys".SimulationDevice, Alarm := #Alarm.Fan, MotorSts =>, Contactor => #DataOut.Fan)
   END_RUNG
   // the same network as SCL:
   #M_MotorFan(FdbkRunning := #DataIn.Fbk_Fan,   // "Motor"
               FeedbackTimeout := T#1s,
               Simulation := "Sys".SimulationDevice,
               Alarm := #Alarm.Fan,
               Contactor => #DataOut.Fan);
END_REGION

REGION Network 31: <<<< FINAL >>>>
   Label( FINAL )
   RUNG wire#powerrail
      Coil( #"NOP" )
   END_RUNG
   // the same network as SCL:
   FINAL:
   #"NOP" := TRUE;
END_REGION

REGION Network 32: Machine is standstill
   RUNG wire#powerrail
      Contact( #Ax.Sts.AxisSts.Standstill )
      wire#w1
      Coil( #Sts.IsStandstill )
   END_RUNG
   RUNG wire#powerrail
      Contact( #DSI.DevicesInSafeState )
   END_RUNG wire#w1
   // the same network as SCL:
   #Sts.IsStandstill := #Ax.Sts.AxisSts.Standstill OR #DSI.DevicesInSafeState;
END_REGION

REGION Network 33: Delay no pending commands
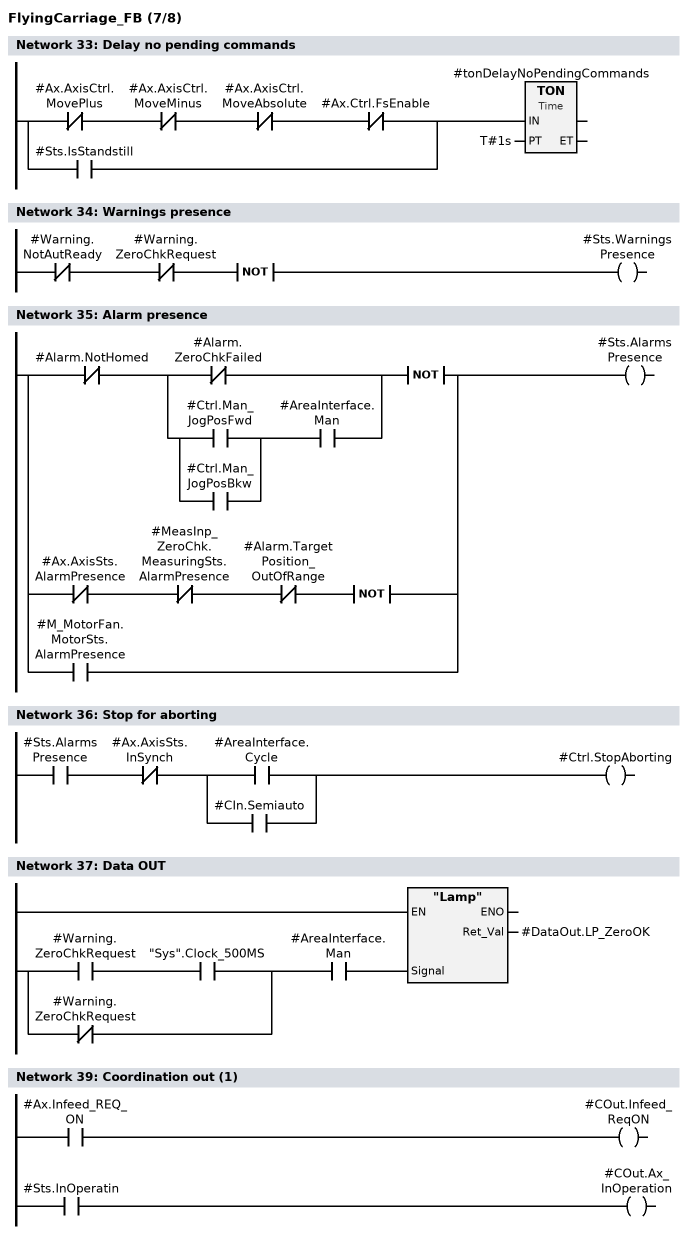
   RUNG wire#powerrail
      I_Contact( #Ax.AxisCtrl.MovePlus )
      I_Contact( #Ax.AxisCtrl.MoveMinus )
      I_Contact( #Ax.AxisCtrl.MoveAbsolute )
      I_Contact( #Ax.Ctrl.FsEnable )
      wire#w1
      { S7_Templates := "time_type := Time" } #tonDelayNoPendingCommands.TON(pt := T#1s, et =>)
   END_RUNG
   RUNG wire#powerrail
      Contact( #Sts.IsStandstill )
   END_RUNG wire#w1
   // the same network as SCL:
   #tonDelayNoPendingCommands.TON(IN := (NOT #Ax.AxisCtrl.MovePlus AND NOT #Ax.AxisCtrl.MoveMinus AND NOT #Ax.AxisCtrl.MoveAbsolute AND NOT #Ax.Ctrl.FsEnable) OR #Sts.IsStandstill,
                           PT := T#1s);
END_REGION

REGION Network 34: Warnings presence
   RUNG wire#powerrail
      I_Contact( #Warning.NotAutReady )
      I_Contact( #Warning.ZeroChkRequest )
      Not()
      Coil( #Sts.WarningsPresence )
   END_RUNG
   // the same network as SCL:
   #Sts.WarningsPresence := NOT (NOT #Warning.NotAutReady AND NOT #Warning.ZeroChkRequest);
END_REGION

REGION Network 35: Alarm presence
   RUNG wire#powerrail
      I_Contact( #Alarm.NotHomed )
      wire#w1
      I_Contact( #Alarm.ZeroChkFailed )
      wire#w2
      Not()
      wire#w4
      Coil( #Sts.AlarmsPresence )
   END_RUNG
   RUNG wire#w1
      Contact( #Ctrl.Man_JogPosFwd )
      wire#w3
      Contact( #AreaInterface.Man )
   END_RUNG wire#w2
   RUNG wire#w1
      Contact( #Ctrl.Man_JogPosBkw )
   END_RUNG wire#w3
   RUNG wire#powerrail
      I_Contact( #Ax.AxisSts.AlarmPresence )
      I_Contact( #MeasInp_ZeroChk.MeasuringSts.AlarmPresence )
      I_Contact( #Alarm.TargetPosition_OutOfRange )
      Not()
   END_RUNG wire#w4
   RUNG wire#powerrail
      Contact( #M_MotorFan.MotorSts.AlarmPresence )
   END_RUNG wire#w4
   // the same network as SCL:
   #Sts.AlarmsPresence := NOT (NOT #Alarm.NotHomed AND (NOT #Alarm.ZeroChkFailed OR ((#Ctrl.Man_JogPosFwd OR #Ctrl.Man_JogPosBkw) AND #AreaInterface.Man))) OR NOT (NOT #Ax.AxisSts.AlarmPresence AND NOT #MeasInp_ZeroChk.MeasuringSts.AlarmPresence AND NOT #Alarm.TargetPosition_OutOfRange) OR #M_MotorFan.MotorSts.AlarmPresence;
END_REGION

REGION Network 36: Stop for aborting
   RUNG wire#powerrail
      Contact( #Sts.AlarmsPresence )
      I_Contact( #Ax.AxisSts.InSynch )
      wire#w1
      Contact( #AreaInterface.Cycle )
      wire#w2
      Coil( #Ctrl.StopAborting )
   END_RUNG
   RUNG wire#w1
      Contact( #CIn.Semiauto )
   END_RUNG wire#w2
   // the same network as SCL:
   #Ctrl.StopAborting := #Sts.AlarmsPresence AND NOT #Ax.AxisSts.InSynch AND (#AreaInterface.Cycle OR #CIn.Semiauto);
END_REGION

REGION Network 37: Data OUT
   RUNG wire#powerrail
      "Lamp"(Signal := wire#w2, Ret_Val => #DataOut.LP_ZeroOK)
   END_RUNG
   RUNG wire#powerrail
      Contact( #Warning.ZeroChkRequest )
      Contact( "Sys".Clock_500MS )
      wire#w1
      Contact( #AreaInterface.Man )
   END_RUNG wire#w2
   RUNG wire#powerrail
      I_Contact( #Warning.ZeroChkRequest )
   END_RUNG wire#w1
   // the same network as SCL:
   #DataOut.LP_ZeroOK := "Lamp"(Signal := ((#Warning.ZeroChkRequest AND "Sys".Clock_500MS) OR NOT #Warning.ZeroChkRequest) AND #AreaInterface.Man);
END_REGION

REGION Network 38 (SCL): Collect machine to area interface
   // Status Motion standtill
   #MachineInterface.MotionsStandStill := #Sts.IsStandstill AND #tonDelayNoPendingCommands.Q;
   // Status machine ready
   #MachineInterface.AutReady := #AreaInterface.Aut
   AND NOT #Sts.AlarmsPresence
   AND NOT #Warning.ZeroChkRequest;

   // Status machine aborting
   #MachineInterface.Aborting := #Ctrl.StopAborting;
   // Status Ack Stop in phase
   #MachineInterface.AckStopInPhase := #Ctrl.StopInPhase AND #MachineInterface.MotionsStandStill;
   // Status Ack Stop programmed
   #MachineInterface.AckStopProgrammed := #Ctrl.StopProgrammed AND #MachineInterface.MotionsStandStill;
   // Status Alarm presence
   #MachineInterface.AlarmsPresence := #Sts.AlarmsPresence;
   // Status Warning presence
   #MachineInterface.WarningPresence := #Sts.WarningsPresence;

   // Warning machine not automatic ready
   IF #AreaInterface.CheckAutReady AND NOT #MachineInterface.AutReady THEN
       #Warning.NotAutReady := TRUE;
   END_IF;
END_REGION

REGION Network 39: Coordination out (1)
   RUNG wire#powerrail
      Contact( #Ax.Infeed_REQ_ON )
      Coil( #COut.Infeed_ReqON )
   END_RUNG
   RUNG wire#powerrail
      Contact( #Sts.InOperatin )
      Coil( #COut.Ax_InOperation )
   END_RUNG
   // the same network as SCL:
   #COut.Infeed_ReqON := #Ax.Infeed_REQ_ON;
   #COut.Ax_InOperation := #Sts.InOperatin;
END_REGION

REGION Network 40: Coordination out (2)
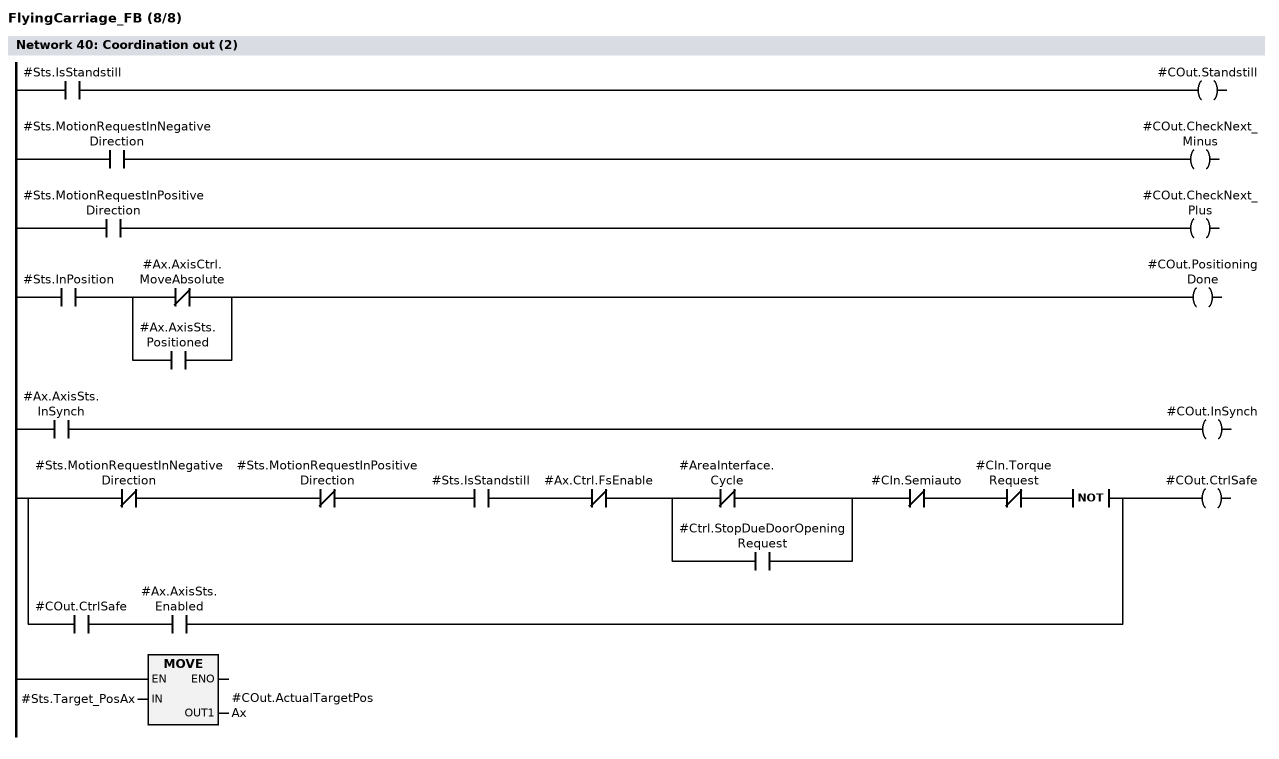
   RUNG wire#powerrail
      Contact( #Sts.IsStandstill )
      Coil( #COut.Standstill )
   END_RUNG
   RUNG wire#powerrail
      Contact( #Sts.MotionRequestInNegativeDirection )
      Coil( #COut.CheckNext_Minus )
   END_RUNG
   RUNG wire#powerrail
      Contact( #Sts.MotionRequestInPositiveDirection )
      Coil( #COut.CheckNext_Plus )
   END_RUNG
   RUNG wire#powerrail
      Contact( #Sts.InPosition )
      wire#w1
      I_Contact( #Ax.AxisCtrl.MoveAbsolute )
      wire#w2
      Coil( #COut.PositioningDone )
   END_RUNG
   RUNG wire#w1
      Contact( #Ax.AxisSts.Positioned )
   END_RUNG wire#w2
   RUNG wire#powerrail
      Contact( #Ax.AxisSts.InSynch )
      Coil( #COut.InSynch )
   END_RUNG
   RUNG wire#powerrail
      I_Contact( #Sts.MotionRequestInNegativeDirection )
      I_Contact( #Sts.MotionRequestInPositiveDirection )
      Contact( #Sts.IsStandstill )
      I_Contact( #Ax.Ctrl.FsEnable )
      wire#w3
      I_Contact( #AreaInterface.Cycle )
      wire#w4
      I_Contact( #CIn.Semiauto )
      I_Contact( #CIn.TorqueRequest )
      Not()
      wire#w5
      Coil( #COut.CtrlSafe )
   END_RUNG
   RUNG wire#w3
      Contact( #Ctrl.StopDueDoorOpeningRequest )
   END_RUNG wire#w4
   RUNG wire#powerrail
      Contact( #COut.CtrlSafe )
      Contact( #Ax.AxisSts.Enabled )
   END_RUNG wire#w5
   RUNG wire#powerrail
      Move(in := #Sts.Target_PosAx, out1 => #COut.ActualTargetPosAx)
   END_RUNG
   // the same network as SCL:
   #COut.Standstill := #Sts.IsStandstill;
   #COut.CheckNext_Minus := #Sts.MotionRequestInNegativeDirection;
   #COut.CheckNext_Plus := #Sts.MotionRequestInPositiveDirection;
   #COut.PositioningDone := #Sts.InPosition AND (NOT #Ax.AxisCtrl.MoveAbsolute OR #Ax.AxisSts.Positioned);
   #COut.InSynch := #Ax.AxisSts.InSynch;
   #COut.CtrlSafe := NOT (NOT #Sts.MotionRequestInNegativeDirection AND NOT #Sts.MotionRequestInPositiveDirection AND #Sts.IsStandstill AND NOT #Ax.Ctrl.FsEnable AND (NOT #AreaInterface.Cycle OR #Ctrl.StopDueDoorOpeningRequest) AND NOT #CIn.Semiauto AND NOT #CIn.TorqueRequest) OR (#COut.CtrlSafe AND #Ax.AxisSts.Enabled);
   #COut.ActualTargetPosAx := #Sts.Target_PosAx;
END_REGION

REGION Network 41 (SCL): HMI
   #HMI.PositionNorm   :=  LREAL_TO_REAL((#TO_Carriage.ActualPosition - #TO_Carriage.PositionLimits_SW.MinPosition)
                          / (#TO_Carriage.PositionLimits_SW.MaxPosition - #TO_Carriage.PositionLimits_SW.MinPosition));
END_REGION
END_FUNCTION_BLOCK
